TEXTLIST TextList_SafetyGuarderrorid
  0 = 'no_error'
  1 = 'not_connected'
  2 = 'invalid_state'
  4 = 'emergency_error'
  8 = 'interlock_error'
  16 = 'shuttle_crash_error'
  32 = 'limit_switch_error'
  64 = 'io_error'
  128 = 'unknown_error'
   = ''
END_TEXTLIST

(* stored: Version 1.1.0.1, ProductVersion 3.1.4024.11
   TextList TextList_SafetyGuarderrorid: Id {1baa04bb-8181-4b8c-879b-14d2a9272b81} *)
